(* IEC 61131-3 sources: SHU_NSTV/CodeSys_Project/Lib/Interfaces, 1 file *)

(* ---- BasicControlCommands.st ---- *)
INTERFACE BasicControlCommands

METHOD Start
VAR_INPUT
	access : BOOL;
	device : BasicControl;
END_VAR

METHOD Stop
VAR_INPUT
	access: BOOL;
	device : BasicControl;
END_VAR
